FUNCTION_BLOCK DataPanel_FREQ_SAE_J1939 (* Frequency/Counter Inputs 7A-8A Status *)
  (* Standard: SAE J1939; Description: Copyright (c) 2026 HR Agrartechnik GmbH *)
  (* Version 1.0, 2026-01-16, generated, HR Agrartechnik GmbH *)
  PACKAGE DataPanel::Status;
  IMPORT DataPanel::io::MI::const::MI;
  IMPORT eclipse4diac::core::TypeHash;
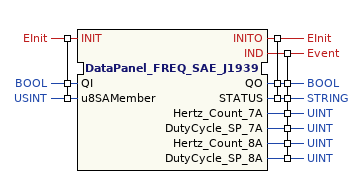
  EVENT_INPUT
    INIT : EInit WITH QI, u8SAMember; (* Service Initialization *)
  END_EVENT
  EVENT_OUTPUT
    INITO : EInit WITH QO, STATUS; (* Initialization Confirm *)
    IND WITH QO, STATUS, Hertz_Count_7A, DutyCycle_SP_7A, Hertz_Count_8A, DutyCycle_SP_8A; (* Indication from Resource *)
  END_EVENT
  VAR_INPUT
    QI : BOOL; (* Event Input Qualifier *)
    u8SAMember : USINT := MI::MI_00; (* Node SA 224..239 *)
  END_VAR
  VAR_OUTPUT
    QO : BOOL; (* Event Output Qualifier *)
    STATUS : STRING; (* Service Status *)
    Hertz_Count_7A : UINT; (* Frequency (Hz) or Count for Input 7A *)
    DutyCycle_SP_7A : UINT; (* Duty Cycle or Setpoint for Input 7A *)
    Hertz_Count_8A : UINT; (* Frequency (Hz) or Count for Input 8A *)
    DutyCycle_SP_8A : UINT; (* Duty Cycle or Setpoint for Input 8A *)
  END_VAR
END_FUNCTION_BLOCK
